// TIA Portal V19 export
TYPE "C904_VAR_IF_PMP_TYPIC"
   STRUCT
      STS_AAN { ExternalAccessible := 'False'; ExternalVisible := 'False'; ExternalWritable := 'False'} : Bool;   // Pomp draait
      BMO_HAND { ExternalAccessible := 'False'; ExternalVisible := 'False'; ExternalWritable := 'False'} : Bool;   // Pomp in hand geschakeld
      TYD_TOT_AAN { ExternalAccessible := 'False'; ExternalVisible := 'False'; ExternalWritable := 'False'} : LInt;   // Totaal aantal draaiuren
      TYD_TOT_AAN_UUR { ExternalAccessible := 'False'; ExternalVisible := 'False'; ExternalWritable := 'False'} : LInt;   // Totaal aantal draaiuren
      TYD_AAN { ExternalAccessible := 'False'; ExternalVisible := 'False'; ExternalWritable := 'False'} : Int;   // Aantal seconden dat pomp aangeschakeld is
      TYD_UIT { ExternalAccessible := 'False'; ExternalVisible := 'False'; ExternalWritable := 'False'} : Int;   // Aantal seconden dat pomp uitgeschakeld is
      ENE_MWA1 { ExternalAccessible := 'False'; ExternalVisible := 'False'; ExternalWritable := 'False'} : Real;   // Stroommeting fase 1
      ENE_MWA2 { ExternalAccessible := 'False'; ExternalVisible := 'False'; ExternalWritable := 'False'} : Real;   // Stroommeting fase 2
      ENE_MWA3 { ExternalAccessible := 'False'; ExternalVisible := 'False'; ExternalWritable := 'False'} : Real;   // Stroommeting fase 3
      EXT_AUT { ExternalAccessible := 'False'; ExternalVisible := 'False'; ExternalWritable := 'False'} : Bool;   // Externe (hoofd) beveiliging aangesproken
      EXT_HW { ExternalAccessible := 'False'; ExternalVisible := 'False'; ExternalWritable := 'False'} : Bool;   // Sturings hardware (PLC) in storing
      STO { ExternalAccessible := 'False'; ExternalVisible := 'False'; ExternalWritable := 'False'} : Struct   // Opsomming van alle storingen
         A001 : Bool;   // Beveiliging aangesproken
         A002 : Bool;   // Storing van de motorbeveiliging van de pomp
         A003 : Bool;   // Storing motorlade
         A004 : Bool;   // Te hoge temperatuur in de motorwikkelingen
         A005 : Bool;   // Fout stroommeting fase 1
         A006 : Bool;   // Fout stroommeting fase 2
         A007 : Bool;   // Fout stroommeting fase 3
         A008 : Bool;   // Droogloop beveiliging actief: LLW vlotter bovenwater
         A009 : Bool;   // Lekdetectie pomp
         A010 : Bool;   // Motorlade uitgeschakeld
         A011 : Bool;   // Motorlade in test
         A012 : Bool;   // Motorlade uitgereden
         AT01 : Bool;   // Discordantie motor: terugmelding niet ontvangen
         AT02 : Bool;   // Discordantie motor: terugmelding blijft aanwezig
         M001 : Bool;   // Werkschakelaar uitgeschakeld
         M002 : Bool;   // Melding: Pomp heeft te lang niet gedraaid. Periodiek onderhoud nodig
      END_STRUCT;
   END_STRUCT;
END_TYPE
